FUNCTION_BLOCK WithInputs (* Only UPDATE updates the data inputs *)
  (* Standard: 61499-2 *)
  (* Version 1.0, 2023-03-07, AK115394 *)
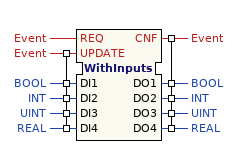
  EVENT_INPUT
    REQ;
    UPDATE WITH DI1, DI2, DI3, DI4;
  END_EVENT
  EVENT_OUTPUT
    CNF WITH DO1, DO3, DO2, DO4;
  END_EVENT
  VAR_INPUT
    DI1 : BOOL := 1;
    DI2 : INT := -10;
    DI3 : UINT := 15;
    DI4 : REAL := 2.0;
  END_VAR
  VAR_OUTPUT
    DO1 : BOOL;
    DO2 : INT;
    DO3 : UINT;
    DO4 : REAL;
  END_VAR
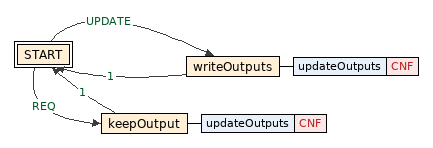
  EC_STATES
    START; (* Initial State *)
    writeOutputs : updateOutputs -> CNF;
    keepOutput : updateOutputs -> CNF;
  END_STATES
  EC_TRANSITIONS
    writeOutputs TO START := 1;
    START TO writeOutputs := UPDATE;
    START TO keepOutput := REQ;
    keepOutput TO START := 1;
  END_TRANSITIONS
  ALGORITHM updateOutputs IN ST:
DO1 := DI1;
DO2 := DI2;
DO3 := DI3;
DO4 := DI4;
  END_ALGORITHM
END_FUNCTION_BLOCK
